// TIA Portal V17 export
// export: Created 2024-08-29T18:23:47.8641845Z, ExportSetting WithDefaults, DisplayName Totally Integrated Automation Portal, DisplayVersion V17 Update 7, DisplayName TIA Portal Openness, DisplayVersion V17 Update 7, DisplayName TIA Portal Version Control Interface, DisplayVersion V17, DisplayName SINAMICS Startdrive Advanced, DisplayVersion V17 SP2, DisplayName SINAMICS Startdrive G110M, G120, G120C, G120D, G120P, G115D, DisplayVersion V17 SP2, DisplayName SINAMICS Startdrive G130, G150, S120, S150, SINAMICS MV, S210, DisplayVersion V17 SP2, DisplayName STEP 7 Professional, DisplayVersion V17 Update 7, DisplayName STEP 7 Safety, DisplayVersion V17 Update 6, DisplayName WinCC Advanced / Unified PC, DisplayVersion V17 Update 7
DATA_BLOCK "FC_IJCORE_MAIN_DB"   // DB1000
VERSION : 0.1
// stored: AutoNumber false, DBAccessibleFromOPCUA true, DBAccessibleFromWebserver true, InstanceOfName FC_IJCORE_MAIN, InstanceOfType FB
"FC_IJCORE_MAIN"
   // VAR
   //    Enable : Bool := TRUE;
   //    Mode : Int := 1;
   //    Indicator : Int := 1;
   //    AlarmReset : Bool := TRUE;
   //    NFP : Array[1..5] of String[30];
   //    AWK : "FB_IJC_AWAKE_SIGNAL";
   //    MSG : Array[1..20] of "FB_IJC_PROTOCOL";
   //    Faults : Array[0..1] of Word;
   // END_VAR
BEGIN
   NFP[1..5] := '';
   AWK.ack_error := TRUE;
   AWK.State_com := 1;
   AWK.T1PresetValue := T#1S;
   AWK.T2PresetValue := T#1M;
   AWK.AwSignalTimeOutFault := FALSE;
   AWK.Reset_Counters := FALSE;
   AWK.Restart_Counter_bit_of_life := 4;
   AWK.NB_Bit_of_Life := FALSE;
   AWK.number_restart := 21346;
   AWK.check_restart := TRUE;
   AWK."Timer"[1].PT := T#1S;
   AWK."Timer"[2].PT := T#2S;
   AWK."Timer"[3].PT := T#200MS;
   AWK."Timer"[4].PT := T#1M;
   AWK."Timer"[5].PT := T#0MS;
   AWK."Timer"[1..3].IN := FALSE;
   AWK."Timer"[4].IN := TRUE;
   AWK."Timer"[5].IN := FALSE;
   MSG[1].MessageType := 'NFP';
   MSG[2..4].MessageType := 'TRC';
   MSG[5].MessageType := 'TRI';
   MSG[6..8].MessageType := 'CNF';
   MSG[9..20].MessageType := '';
   MSG[1].MessageNumber := 1;
   MSG[2].MessageNumber := 2;
   MSG[3].MessageNumber := 3;
   MSG[4].MessageNumber := 4;
   MSG[5].MessageNumber := 5;
   MSG[6].MessageNumber := 6;
   MSG[7].MessageNumber := 7;
   MSG[8].MessageNumber := 8;
   MSG[9..20].MessageNumber := 0;
   MSG[1..8].TraceabilityMode := 1;
   MSG[9..20].TraceabilityMode := 0;
   MSG[1..20].SendMessage := FALSE;
   MSG[1].MasterNFP := FALSE;
   MSG[2].MasterNFP := TRUE;
   MSG[3..20].MasterNFP := FALSE;
   MSG[1..20].NFP := '';
   MSG[1..20].Scan := '';
   MSG[1..20].KANBAN := '';
   MSG[1..20].ScrewTorqueInt := 16#0000;
   MSG[1..20].ScrewTorqueFloat := 16#0000;
   MSG[1..20].ScrewAngle := 16#0000;
   MSG[1..20].ProcessStatus := 0;
   MSG[1..8].ErrReset := TRUE;
   MSG[9..20].ErrReset := FALSE;
   MSG[1..20].oNFP := '';
   MSG[1..20].MessageDone := FALSE;
   MSG[1..20].Answer := 0;
   MSG[1..20].Fault := 0;
   MSG[1..8].State := 10;
   MSG[9..20].State := 0;
   MSG[1].SEND_OFFSET.SW := 4;
   MSG[2].SEND_OFFSET.SW := 6;
   MSG[3].SEND_OFFSET.SW := 8;
   MSG[4].SEND_OFFSET.SW := 10;
   MSG[5].SEND_OFFSET.SW := 12;
   MSG[6].SEND_OFFSET.SW := 14;
   MSG[7].SEND_OFFSET.SW := 16;
   MSG[8].SEND_OFFSET.SW := 18;
   MSG[9..20].SEND_OFFSET.SW := 0;
   MSG[1].SEND_OFFSET.MSG := 604;
   MSG[2].SEND_OFFSET.MSG := 684;
   MSG[3].SEND_OFFSET.MSG := 764;
   MSG[4].SEND_OFFSET.MSG := 844;
   MSG[5].SEND_OFFSET.MSG := 924;
   MSG[6].SEND_OFFSET.MSG := 1004;
   MSG[7].SEND_OFFSET.MSG := 1084;
   MSG[8].SEND_OFFSET.MSG := 1164;
   MSG[9..20].SEND_OFFSET.MSG := 0;
   MSG[1].REC_OFFSET.SW := 0;
   MSG[2].REC_OFFSET.SW := 2;
   MSG[3].REC_OFFSET.SW := 4;
   MSG[4].REC_OFFSET.SW := 6;
   MSG[5].REC_OFFSET.SW := 8;
   MSG[6].REC_OFFSET.SW := 10;
   MSG[7].REC_OFFSET.SW := 12;
   MSG[8].REC_OFFSET.SW := 14;
   MSG[9..20].REC_OFFSET.SW := 0;
   MSG[1].REC_OFFSET.MSG := 602;
   MSG[2].REC_OFFSET.MSG := 634;
   MSG[3].REC_OFFSET.MSG := 666;
   MSG[4].REC_OFFSET.MSG := 698;
   MSG[5].REC_OFFSET.MSG := 730;
   MSG[6].REC_OFFSET.MSG := 762;
   MSG[7].REC_OFFSET.MSG := 794;
   MSG[8].REC_OFFSET.MSG := 826;
   MSG[9..20].REC_OFFSET.MSG := 0;
   MSG[1].REC_OFFSET.ANS := 600;
   MSG[2].REC_OFFSET.ANS := 632;
   MSG[3].REC_OFFSET.ANS := 664;
   MSG[4].REC_OFFSET.ANS := 696;
   MSG[5].REC_OFFSET.ANS := 728;
   MSG[6].REC_OFFSET.ANS := 760;
   MSG[7].REC_OFFSET.ANS := 792;
   MSG[8].REC_OFFSET.ANS := 824;
   MSG[9..20].REC_OFFSET.ANS := 0;
   MSG[1].ONS[1..8] := FALSE;
   MSG[2].ONS[1..8] := FALSE;
   MSG[3].ONS[1..8] := FALSE;
   MSG[4].ONS[1..8] := FALSE;
   MSG[5].ONS[1..8] := FALSE;
   MSG[6].ONS[1..8] := FALSE;
   MSG[7].ONS[1..8] := FALSE;
   MSG[8].ONS[1..8] := FALSE;
   MSG[9].ONS[1..8] := FALSE;
   MSG[10].ONS[1..8] := FALSE;
   MSG[11].ONS[1..8] := FALSE;
   MSG[12].ONS[1..8] := FALSE;
   MSG[13].ONS[1..8] := FALSE;
   MSG[14].ONS[1..8] := FALSE;
   MSG[15].ONS[1..8] := FALSE;
   MSG[16].ONS[1..8] := FALSE;
   MSG[17].ONS[1..8] := FALSE;
   MSG[18].ONS[1..8] := FALSE;
   MSG[19].ONS[1..8] := FALSE;
   MSG[20].ONS[1..8] := FALSE;
   Faults[0..1] := 16#0000;
END_DATA_BLOCK
